FUNCTION_BLOCK OvenBasic
VAR
	_HeatCommand: HeatCommand;
	_Temp : REAL;
	_TempSetPoint : REAL;
END_VAR

METHOD Cyclic : BOOL
//cmd := HeatCommand;
IF _HeatCommand.Consume THEN
	TempSetPoint := _HeatCommand.TempSetPoint; //set the oven temp set point
END_IF

regulateTemp();

IF Temp = TempSetPoint THEN
	_HeatCommand.Finished();//report status when command is done
END_IF

_HeatCommand.Execute := 0;
END_METHOD

METHOD regulateTemp : BOOL
VAR_INPUT
END_VAR
//warm up/cool down over time
IF Temp < TempSetPoint THEN
	Temp := Temp + 1;
ELSIF Temp > TempSetPoint THEN
	Temp := Temp - 1;
END_IF

regulateTemp := Temp = TempSetPoint;
END_METHOD

METHOD StartHeating : BOOL
VAR_INPUT
	temp : REAL;
	status: IPLCopenCall;
END_VAR
_HeatCommand.TempSetPoint := temp;

IF status = 0 THEN
	_HeatCommand.Execute := 1;
ELSE
	status.Start(_HeatCommand);
END_IF
END_METHOD

PROPERTY Temp : REAL
GET
Temp := _Temp;
END_GET
SET
_Temp := Temp;
END_SET
END_PROPERTY

PROPERTY TempSetPoint : REAL
GET
TempSetPoint := _TempSetPoint;
END_GET
SET
_TempSetPoint := TempSetPoint;
END_SET
END_PROPERTY

END_FUNCTION_BLOCK

(* stored: Version 1.1.0.1
   POU OvenBasic: Id {f06dffbc-4722-072d-2af9-eca0de705433}, SpecialFunc None
   Method Cyclic: Id {cadd8092-5caa-0878-1061-812a85cdf4f3}
   Method regulateTemp: Id {e7b4fd20-002e-0a00-2400-c893399805ba}
   Method StartHeating: Id {4682e446-3b47-0d83-307f-2a9af1f7b249}
   Property Temp: Id {8402adfa-4656-07d8-31e0-c7336fe48348}
   Get Get: Id {42a4bc8c-c843-049d-0017-e2a236bdaf56}
   Set Set: Id {e439bc0f-f6df-0042-3b99-ff0e48f51203}
   Property TempSetPoint: Id {72a1bc95-d7ae-06b1-349a-14c2e0298e28}
   Get Get: Id {8fcf468c-17ca-0c09-27b2-079b919c78e2}
   Set Set: Id {a23980ee-440c-0f77-3e3b-5060688a1c12} *)
